Staubli VAL3: TP1_Paolo.dtx

frame fTable = {x=544.793496, y=2.880447, z=-170.95, rx=-179.999977, ry=-0.0003, rz=0.000308, fatherId=world[0]}
jointRx j0
jointRx jDepart = {j1=-7.215316, j2=54.432296, j3=135.763663, j4=-6.983157, j5=-101.065649, j6=-91.233508}
mdesc mPriseDepose = {vel=5}
mdesc mRapide100joint = {vel=25}
pointRx pDepose[2]
  [0] = {x=80.895535, y=164.405443, z=205.485609, rx=20.949006, ry=91.010648, rz=69.047818, fatherId=fTable[0]}
  [1] = {x=83.817549, y=-298.865741, z=205.487219, rx=20.949006, ry=91.010648, rz=69.047818, fatherId=fTable[0]}
pointRx pPrise = {x=81.971792, y=-6.229802, z=205.486202, rx=20.949006, ry=91.010648, rz=69.047818, fatherId=fTable[0]}
sio sData = {link=Socket\staubli_server}
tool tPince = {x=-1.667681, y=-1.981137, z=74.877299, rx=0, ry=0, rz=0, fatherId=flange[0], ioLink=valve1}
trsf trApproZ = {z=-50}
